{attribute 'GeneratedUsingTerminal: EL6201-0000-0017'}
{attribute addProperty BoxType "EL6201-0000-0017"}
{attribute addProperty Id "Slave_16A_DI0BOOL1Slave_16A_DI1BOOL1Slave_16A_DI2BOOL1Slave_16A_DI3BOOL1Slave_16B_DI0BOOL1Slave_16B_DI1BOOL1Slave_16B_DI2BOOL1Slave_16B_DI3BOOL1"}
{attribute addProperty CRC "3775625583"}
{attribute addProperty Size "8"}
TYPE Slave_16_Inputs_E10B796F :
STRUCT
	{attribute addProperty Name "Slave_16A_DI0"}
	Slave_16A_DI0 : BOOL;
	{attribute addProperty Name "Slave_16A_DI1"}
	Slave_16A_DI1 : BOOL;
	{attribute addProperty Name "Slave_16A_DI2"}
	Slave_16A_DI2 : BOOL;
	{attribute addProperty Name "Slave_16A_DI3"}
	Slave_16A_DI3 : BOOL;
	{attribute addProperty Name "Slave_16B_DI0"}
	Slave_16B_DI0 : BOOL;
	{attribute addProperty Name "Slave_16B_DI1"}
	Slave_16B_DI1 : BOOL;
	{attribute addProperty Name "Slave_16B_DI2"}
	Slave_16B_DI2 : BOOL;
	{attribute addProperty Name "Slave_16B_DI3"}
	Slave_16B_DI3 : BOOL;
END_STRUCT
END_TYPE

(* stored: Version 1.2.0.0, ProductVersion 3.1.4024.11
   DUT Slave_16_Inputs_E10B796F: Id {d9da7022-866c-4f68-855a-b98152aa3d4e} *)
